// TIA Portal V20 export
DATA_BLOCK "Alarms"   // DB149
// stored: Access Published, MemoryReserve 100, Namespace Unit1
   VAR
      unitAlarms { ExternalWritable := 'False'} : "LAF_typeAlarms";
      emAlarms { ExternalWritable := 'False'} : Array[0.._.U1_NO_OF_EMs] of "LAF_typeAlarms";
      maintenanceFaults { ExternalWritable := 'False'} : Array[0..199] of Bool;   // PFE Maintenance Faults
      productionFaults { ExternalWritable := 'False'} : Array[0..199] of Bool;   // PFE Production Faults
      toolingFault { ExternalWritable := 'False'} : Array[0..199] of Bool;   // PFE Tooling Faults
      qualityFault { ExternalWritable := 'False'} : Array[0..199] of Bool;   // PFE Quality Faults
      throughputFaultBlocked { ExternalWritable := 'False'} : Array[0..199] of Bool;   // PFE Throughput Fault Blocked
      throughputFaultStarved { ExternalWritable := 'False'} : Array[0..199] of Bool;   // PFE Throughput Fault Starved
      throughputFault { ExternalWritable := 'False'} : Array[0..199] of Bool;   // PFE Throughput Fault
      systemFaultGeneral { ExternalWritable := 'False'} : Array[0..199] of Bool;   // PFE System Fault General
      materialFault { ExternalWritable := 'False'} : Array[0..199] of Bool;   // PFE Material Fault
      maintenanceWarnings { ExternalWritable := 'False'} : Array[0..199] of Bool;   // PFE Maintenance Warnings
      productionWarning { ExternalWritable := 'False'} : Array[0..199] of Bool;   // PFE Production Warning
      toolingWarning { ExternalWritable := 'False'} : Array[0..199] of Bool;   // PFE Tooling Warning
      qualityWarning { ExternalWritable := 'False'} : Array[0..199] of Bool;   // PFE Quality Warning
      throughputWarning { ExternalWritable := 'False'} : Array[0..199] of Bool;   // PFE Throughput Warning
      systemWarning { ExternalWritable := 'False'} : Array[0..199] of Bool;   // PFE System Warning
      materialWarning { ExternalWritable := 'False'} : Array[0..199] of Bool;   // PFE Material Warning
      maintenanceStatus { ExternalWritable := 'False'} : Array[0..199] of Bool;   // PFE Maintenance Status
      productionStatus { ExternalWritable := 'False'} : Array[0..199] of Bool;   // PFE Production Status
      toolingStatus { ExternalWritable := 'False'} : Array[0..199] of Bool;   // PFE Tooling Status
      qualityStatus { ExternalWritable := 'False'} : Array[0..199] of Bool;   // PFE Quality Status
      throughputStatus { ExternalWritable := 'False'} : Array[0..199] of Bool;   // PFE Throughput Status
      systemStatus { ExternalWritable := 'False'} : Array[0..199] of Bool;   // PFE System Status
      materialStatus { ExternalWritable := 'False'} : Array[0..199] of Bool;   // PFE Material Status
      TonMaintenanceFault { ExternalWritable := 'False'} : Array[0..199] of TON_TIME;   // PFE Maintenance Faults Ton Timer
      TonProductionFault { ExternalWritable := 'False'} : Array[0..199] of TON_TIME;   // PFE Production Faults Ton Timer
      TonToolingFault { ExternalWritable := 'False'} : Array[0..199] of TON_TIME;   // PFE Tooling Faults Ton Timer
      TonQualityFault { ExternalWritable := 'False'} : Array[0..199] of TON_TIME;   // PFE Quality Faults Ton Timer
      TonThroughputFaultBlocked { ExternalWritable := 'False'} : Array[0..199] of TON_TIME;   // PFE Throughput Fault Blocked Ton Timer
      TonThroughputFaultStarved { ExternalWritable := 'False'} : Array[0..199] of TON_TIME;   // PFE Throughput Fault Starved Ton Timer
      TonThroughputFault { ExternalWritable := 'False'} : Array[0..199] of TON_TIME;   // PFE Throughput Fault Ton Timer
      TonSystemFaultGeneral { ExternalWritable := 'False'} : Array[0..199] of TON_TIME;   // PFE System Fault General Ton Timer
      TonMaterialFault { ExternalWritable := 'False'} : Array[0..199] of TON_TIME;   // PFE Material Fault Ton Timer
      TonMaintenanceWarning { ExternalWritable := 'False'} : Array[0..199] of TON_TIME;   // PFE Maintenance Warnings Ton Timer
      TonProductionWarning { ExternalWritable := 'False'} : Array[0..199] of TON_TIME;   // PFE Production Warning Ton Timer
      TonToolingWarning { ExternalWritable := 'False'} : Array[0..199] of TON_TIME;   // PFE Tooling Warning Ton Timer
      TonQualityWarning { ExternalWritable := 'False'} : Array[0..199] of TON_TIME;   // PFE Quality Warning Ton Timer
      TonThroughputWarning { ExternalWritable := 'False'} : Array[0..199] of TON_TIME;   // PFE Throughput Warning Ton Timer
      TonSystemWarning { ExternalWritable := 'False'} : Array[0..199] of TON_TIME;   // PFE System Warning Ton Timer
      TonMaterialWarning { ExternalWritable := 'False'} : Array[0..199] of TON_TIME;   // PFE Material Warning Ton Timer
      TonMaintenanceStatus { ExternalWritable := 'False'} : Array[0..199] of TON_TIME;   // PFE Maintenance Status Ton Timer
      TonProductionStatus { ExternalWritable := 'False'} : Array[0..199] of TON_TIME;   // PFE Production Status Ton Timer
      TonToolingStatus { ExternalWritable := 'False'} : Array[0..199] of TON_TIME;   // PFE Tooling Status Ton Timer
      TonQualityStatus { ExternalWritable := 'False'} : Array[0..199] of TON_TIME;   // PFE Quality Status Ton Timer
      TonThroughputStatus { ExternalWritable := 'False'} : Array[0..199] of TON_TIME;   // PFE Throughput Status Ton Timer
      TonSystemStatus { ExternalWritable := 'False'} : Array[0..199] of TON_TIME;   // PFE System Status Ton Timer
      TonMaterialStatus { ExternalWritable := 'False'} : Array[0..199] of TON_TIME;   // PFE Material Status Ton Timer
   END_VAR
BEGIN
   // maintenanceFaults[0] : EM Error
   // maintenanceFaults[1] : Frame Cover Not Detect
   // maintenanceFaults[2] : All Em Status is not linked
   // maintenanceFaults[10] : 24 Hours Time Over
   // systemFaultGeneral[0] : MotorPowerTripped
   // systemFaultGeneral[1] : ReelcutConveyorRingBlowPowerTripped
   // systemFaultGeneral[2] : Stacking1ConveyorRingBlowPowerTripped
   // systemFaultGeneral[3] : Stacking2ConveyorRingBlowPowerTripped
   // systemFaultGeneral[4] : E6404PwsControllerPowerSmpsAcPowerTripped
   // systemFaultGeneral[5] : E6704PwsControllerPowerSmpsAcPowerTripped
   // systemFaultGeneral[6] : E6804PwsSafetyPowerSmpsAcPowerTripped
   // systemFaultGeneral[7] : PowerMeterPowerTripped
   // systemFaultGeneral[8] : PowerMeterControlPowerTripped
   // systemFaultGeneral[9] : ProcessorPowerOnTripped
   // systemFaultGeneral[10] : ProgrammingPowerOutletTripped
   // systemFaultGeneral[11] : PanelLedPowerTripped
   // systemFaultGeneral[12] : ControlLevelHubPowerTripped
   // systemFaultGeneral[13] : MainHmiPowerTripped
   // systemFaultGeneral[14] : PortableHmiPowerTripped
   // systemFaultGeneral[15] : PortableHmiPowerTripped
   // systemFaultGeneral[16] : 120VacControlPowerTrPrimaryTripped
   // systemFaultGeneral[17] : 120VacControlPowerTrSecondaryTripped
   // systemFaultGeneral[18] : ControlPowerOnTripped
   // systemFaultGeneral[19] : VisionMonitorPowerStripOutletPowerTripped
   // systemFaultGeneral[20] : McuRfidHandyPowerStripOutletPowerTripped
   // systemFaultGeneral[21] : VisionLightControllerPowerStripOutletPowerTripped
   // systemFaultGeneral[22] : FfuPower1PowerTripped
   // systemFaultGeneral[23] : Et200MpIoOutputPowerTripped
   // systemFaultGeneral[24] : JunctionBoxControlPowerTripped
   // systemFaultGeneral[25] : Class2SmpsPowerTripped
   // systemFaultGeneral[26] : Class2SmpsMonitoringTripped
   // systemFaultGeneral[27] : Et200EcoPn1PowerTripped
   // systemFaultGeneral[28] : Et200EcoPn2PowerTripped
   // systemFaultGeneral[29] : Et200EcoPn3PowerTripped
   // systemFaultGeneral[30] : PanelFanPowerTripped
   // systemFaultGeneral[31] : ControllerDcPowerTripped
   // systemFaultGeneral[32] : ServoControlPowerTripped
   // systemFaultGeneral[33] : Manifold1ControlPowerTripped
   // systemFaultGeneral[34] : RfidPowerTripped
   // systemFaultGeneral[35] : QrReaderPowerTripped
   // systemFaultGeneral[36] : QrReaderPowerTripped
   // systemFaultGeneral[37] : ControllerDcPowerTripped
   // systemFaultGeneral[38] : HandyQrReaderPowerTripped
   // systemFaultGeneral[39] : VisionControllerPowerTripped
   // systemFaultGeneral[40] : LineLaserModule1PowerTripped
   // systemFaultGeneral[41] : LineLaserModule2PowerTripped
   // systemFaultGeneral[42] : EpcController1PowerTripped
   // systemFaultGeneral[43] : EpcController2PowerTripped
   // systemFaultGeneral[44] : EpcController3PowerTripped
   // systemFaultGeneral[45] : DriveCliqHubPowerTripped
   // systemFaultGeneral[46] : EquipmentLedPowerTripped
   // systemFaultGeneral[47] : MotorPowerMcCoilPowerTripped
   // systemFaultGeneral[48] : SafetyDcPowerTripped
   // systemFaultGeneral[49] : Et200SpIoSafetyPowerTripped
   // systemFaultGeneral[50] : JunctionBoxControlPowerTripped
   // systemFaultGeneral[51] : Et200EcoPnSafetyT1PowerTripped
   // systemFaultGeneral[52] : MainHMIPowerTrpped
   // systemFaultGeneral[53] : ControlDcPowerTripped
   // systemFaultGeneral[54] : SafetyDcPowerTripped
   // systemFaultGeneral[100] : PlcPowerSmpsDcOk
   // systemFaultGeneral[101] : ControlPowerSmpsDcOk
   // systemFaultGeneral[102] : ControllerPowerSmpsDcOk
   // systemFaultGeneral[103] : ControllerPowerSmpsDcOk
   // systemFaultGeneral[104] : SafetyPowerSmpsDcOk
   // systemFaultGeneral[110] : SLM SinaInfeed Fault
   // systemFaultGeneral[111] : Manifold1 Control Power FeedBack Fault
   // systemFaultGeneral[113] : FFU1 Control Power FeedBack Fault
   // systemFaultGeneral[114] : FFU2 Control Power FeedBack Fault
   // systemFaultGeneral[115] : Main Pressure Switch-1 Fault
   // systemFaultGeneral[116] : Main Pressure Switch-2 Fault
   // maintenanceWarnings[10] : 8 Hours Time Over
END_DATA_BLOCK
